PROGRAM PRG_10_TempHumidAnalytics
VAR
	TempSensor								: GenericSensor;
	HumiditySensor							: GenericSensor;
	
	{attribute 'OPC.UA.DA' := '1'}					// enable/disable to OPC UA
	{attribute 'OPC.UA.DA.Access' := '1'}			// read only
	{attribute 'OPC.UA.DA.StructuredType' := '1'}	// define variable as STRUCT for OPC UA
	TempSensorStruct						: SingleSensor_DataModel;
	
	{attribute 'OPC.UA.DA' := '1'}					// enable/disable to OPC UA
	{attribute 'OPC.UA.DA.Access' := '1'}			// read only
	{attribute 'OPC.UA.DA.StructuredType' := '1'}	// define variable as STRUCT for OPC UA
	HumiditySensorStruct					: SingleSensor_DataModel;
END_VAR

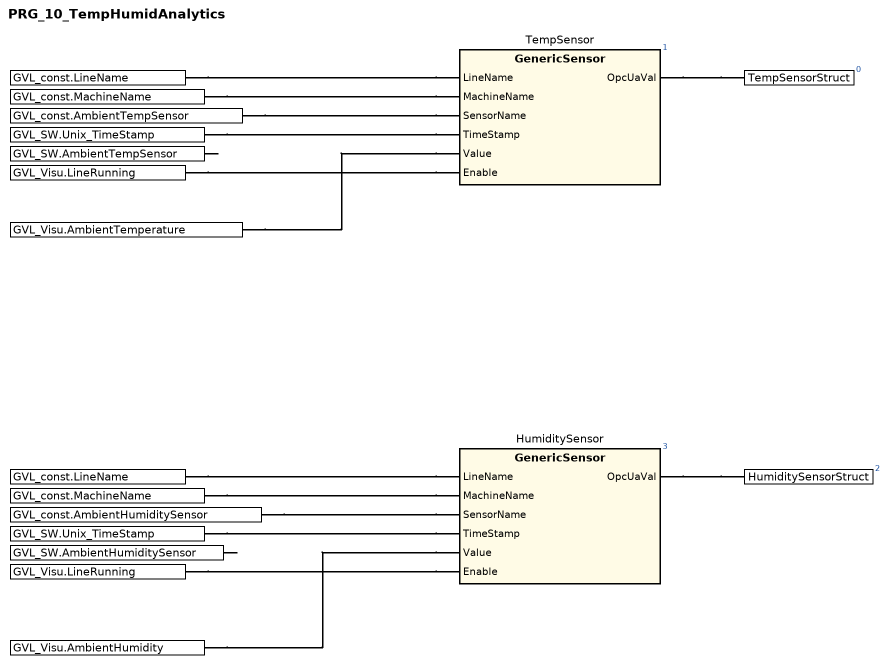
TempSensorStruct := TempSensor.OpcUaVal;
TempSensor(
    LineName := GVL_const.LineName,
    MachineName := GVL_const.MachineName,
    SensorName := GVL_const.AmbientTempSensor,
    TimeStamp := GVL_SW.Unix_TimeStamp,
    Value := GVL_Visu.AmbientTemperature,
    Enable := GVL_Visu.LineRunning); // GenericSensor
HumiditySensorStruct := HumiditySensor.OpcUaVal;
HumiditySensor(
    LineName := GVL_const.LineName,
    MachineName := GVL_const.MachineName,
    SensorName := GVL_const.AmbientHumiditySensor,
    TimeStamp := GVL_SW.Unix_TimeStamp,
    Value := GVL_Visu.AmbientHumidity,
    Enable := GVL_Visu.LineRunning); // GenericSensor
// GVL_SW.AmbientTempSensor: input not connected
// GVL_SW.AmbientHumiditySensor: input not connected

END_PROGRAM

(* stored: Version 1.1.0.1, ProductVersion 3.1.4024.15
   POU PRG_10_TempHumidAnalytics: Id {71aa9778-4091-4bf1-b573-d9e4e399eb71}, SpecialFunc None *)
